Yaskawa INFORM job: GO-TO-STATION-2-BACK.JBI

/JOB
//NAME GO-TO-STATION-2-BACK
//POS
///NPOS 2,0,0,1,0,0
///TOOL 0
///POSTYPE PULSE
///PULSE
C00000=292966,-222014,-26224,0,-132993,69558
C00001=301699,-53771,-35411,94802,-86201,103803
P00000=0,-222014,-26224,0,-132993,0
//INST
///DATE 2018/09/17 10:43
///ATTR SC,RW
///GROUP1 RB1
NOP
MOVJ P0000 VJ=50.00
'*****
SETREG MREG#(1) 1
MOVJ C00000 VJ=25.00
'*****
SETREG MREG#(1) 120
MOVJ C00001 VJ=25.00
'*****
SETREG MREG#(1) 121
END
